   ! RB-1000SAD (Robobel Type):
   !pers tooldata tRB1000SAD_0   := [true,[[181.9,0,472.5],[0.866025,0,0.5,0]],[10,[31,0,260],[1,0,0,0],0,0,0]];
   !pers tooldata tRB1000SAD_100 := [true,[[268.5,0,522.5],[0.866025,0,0.5,0]],[10,[31,0,260],[1,0,0,0],0,0,0]];
   !pers tooldata tRB1000SAD_150 := [true,[[311.8,0,547.5],[0.866025,0,0.5,0]],[10,[31,0,260],[1,0,0,0],0,0,0]];
   !pers tooldata tRB1000SAD_200 := [true,[[355.1,0,572.5],[0.866025,0,0.5,0]],[10,[31,0,260],[1,0,0,0],0,0,0]];
   !pers tooldata tRB1000SAD_250 := [true,[[398.4,0,597.5],[0.866025,0,0.5,0]],[10,[31,0,260],[1,0,0,0],0,0,0]];
   !pers tooldata tRB1000SAD_300 := [true,[[441.7,0,622.5],[0.866025,0,0.5,0]],[10,[31,0,260],[1,0,0,0],0,0,0]];

   ! RB-1000SSD (Robobel Type):
   !PERS tooldata tRB1000SSD_0   := [true,[[181.9,0,472.5],[0.866025,0,0.5,0]],[10,[31,0,260],[1,0,0,0],0,0,0]];
   !PERS tooldata tRB1000SSD_100 := [true,[[268.5,0,522.5],[0.866025,0,0.5,0]],[10,[31,0,260],[1,0,0,0],0,0,0]];
   !PERS tooldata tRB1000SSD_150 := [true,[[311.8,0,547.5],[0.866025,0,0.5,0]],[10,[31,0,260],[1,0,0,0],0,0,0]];
   !PERS tooldata tRB1000SSD_200 := [true,[[355.1,0,572.5],[0.866025,0,0.5,0]],[10,[31,0,260],[1,0,0,0],0,0,0]];
   !PERS tooldata tRB1000SSD_250 := [true,[[398.4,0,597.5],[0.866025,0,0.5,0]],[10,[31,0,260],[1,0,0,0],0,0,0]];
   !PERS tooldata tRB1000SSD_300 := [true,[[441.7,0,622.5],[0.866025,0,0.5,0]],[10,[31,0,260],[1,0,0,0],0,0,0]];



   ! Speed data:
   const speeddata vPaint50   := [50,300,1000,50];
   const speeddata vPaint100  := [100,300,100,100];
   const speeddata vPaint150  := [150,300,150,150];
   const speeddata vPaint200  := [200,300,200,200];
   const speeddata vPaint250  := [250,300,250,250];
   const speeddata vPaint300  := [300,300,300,300];
   const speeddata vPaint350  := [350,300,350,350];
   const speeddata vPaint400  := [400,300,400,400];
   const speeddata vPaint450  := [450,300,450,450];
   const speeddata vPaint500  := [500,300,500,500];
   const speeddata vPaint550  := [550,300,1000,500];
   const speeddata vPaint600  := [600,300,1000,500];
   const speeddata vPaint650  := [650,300,1000,500];
   const speeddata vPaint700  := [700,300,1000,500];
   const speeddata vPaint750  := [750,300,1000,500];
   const speeddata vPaint800  := [800,300,1000,500];
   const speeddata vPaint850  := [850,300,1000,500];
   const speeddata vPaint900  := [900,300,1000,500];
   const speeddata vPaint950  := [950,300,1000,500];
   const speeddata vPaint1000 := [1000,300,1000,500];
   const speeddata vPaint1100 := [1100,300,1000,500];
   const speeddata vPaint1200 := [1200,300,1000,500];
   const speeddata vPaint1300 := [1300,300,1000,500];
   const speeddata vPaint1400 := [1400,300,1000,500];
   const speeddata vPaint1500 := [1500,300,1000,500];
   const speeddata vPaint1600 := [1600,300,1000,500];
   const speeddata vPaint1700 := [1700,300,1000,500];
   const speeddata vPaint1800 := [1800,300,1000,500];
   const speeddata vPaint1900 := [1900,300,1000,500];
   const speeddata vPaint2000 := [2000,300,1000,500];
   const speeddata vPaint2100 := [2100,300,1000,500];
   const speeddata vPaint2200 := [2200,300,1000,500];
   const speeddata vPaint2300 := [2300,300,1000,500];
   const speeddata vPaint2400 := [2400,300,1000,500];
   const speeddata vPaint2500 := [2500,300,1000,500];

   ! Speed data (High Flow Bell):
   const speeddata vHFB50   := [50,150,50,50];
   const speeddata vHFB100  := [100,150,100,100];
   const speeddata vHFB150  := [150,150,150,150];
   const speeddata vHFB200  := [200,150,200,200];
   const speeddata vHFB250  := [250,150,250,250];
   const speeddata vHFB300  := [300,150,300,300];
   const speeddata vHFB350  := [350,150,350,350];
   const speeddata vHFB400  := [400,150,400,400];
   const speeddata vHFB450  := [450,150,450,450];
   const speeddata vHFB500  := [500,150,500,500];
   const speeddata vHFB550  := [550,150,1000,500];
   const speeddata vHFB600  := [600,150,1000,500];
   const speeddata vHFB650  := [650,150,1000,500];
   const speeddata vHFB700  := [700,150,1000,500];
   const speeddata vHFB750  := [750,150,1000,500];
   const speeddata vHFB800  := [800,150,1000,500];
   const speeddata vHFB850  := [850,150,1000,500];
   const speeddata vHFB900  := [900,150,1000,500];
   const speeddata vHFB950  := [950,150,1000,500];
   const speeddata vHFB1000 := [1000,150,1000,500];
   const speeddata vHFB1100 := [1100,150,1000,500];
   const speeddata vHFB1200 := [1200,150,1000,500];
   const speeddata vHFB1300 := [1300,150,1000,500];
   const speeddata vHFB1400 := [1400,150,1000,500];
   const speeddata vHFB1500 := [1500,150,1000,500];
   const speeddata vHFB1600 := [1600,150,1000,500];
   const speeddata vHFB1700 := [1700,150,1000,500];
   const speeddata vHFB1800 := [1800,150,1000,500];
   const speeddata vHFB1900 := [1900,150,1000,500];
   const speeddata vHFB2000 := [2000,150,1000,500];
   const speeddata vHFB2100 := [2100,150,1000,500];
   const speeddata vHFB2200 := [2200,150,1000,500];
   const speeddata vHFB2300 := [2300,150,1000,500];
   const speeddata vHFB2400 := [2400,150,1000,500];
   const speeddata vHFB2500 := [2500,150,1000,500];



   ! Zone data:
   const zonedata zPaint1   := [false,1,1,1,0.15,1,0.15];
   const zonedata zPaint5   := [false,5,8,8,0.8,8,0.8];
   const zonedata zPaint10  := [false,10,15,15,1.5,15,1.5];
   const zonedata zPaint15  := [false,15,23,23,2.3,23,2.3];
   const zonedata zPaint20  := [false,20,30,30,3,30,3];
   const zonedata zPaint30  := [false,30,45,45,4.5,45,4.5];
   const zonedata zPaint40  := [false,40,60,60,6,60,6];
   const zonedata zPaint50  := [false,50,75,75,7.5,75,7.5];
   const zonedata zPaint60  := [false,60,90,90,9,90,9];
   const zonedata zPaint80  := [false,80,120,120,12,120,12];
   const zonedata zPaint100 := [false,100,150,150,15,150,15];
   const zonedata zPaint150 := [false,150,225,225,23,225,23];
   const zonedata zPaint200 := [false,200,300,300,30,300,30];
   const zonedata zPaint250 := [false,250,375,375,37.5,375,37.5];
   const zonedata zPaint300 := [false,300,450,450,45,450,45];



   proc ConfSettingsOff()
      ConfJ \Off;
      ConfL \Off;
   endproc



endmodule

--- Backups/Robo_open_v2/RAPID/TASK1/SYSMOD/sysdata.sys ---
module sysdata(sysmodule)

   ! Warning: Do not remove standard data from this module.

   pers robtarget pHomePos   := [[0,0,0],[9E+09,9E+09,9E+09,9E+09],[-1,-1,1,0],[9E+09,9E+09,9E+09,9E+09,9E+09,9E+09]];
   pers robtarget pMtrlChPos := [[0,0,0],[9E+09,9E+09,9E+09,9E+09],[-1,-1,1,0],[9E+09,9E+09,9E+09,9E+09,9E+09,9E+09]];
   pers robtarget pReadyPos  := [[0,0,0],[9E+09,9E+09,9E+09,9E+09],[-1,-1,1,0],[9E+09,9E+09,9E+09,9E+09,9E+09,9E+09]];
   pers robtarget pUserPos   := [[0,0,0],[9E+09,9E+09,9E+09,9E+09],[-1,-1,1,0],[9E+09,9E+09,9E+09,9E+09,9E+09,9E+09]];

   pers jointtarget jHomePos   := [[9E+09,9E+09,9E+09,9E+09,9E+09,9E+09],[9E+09,9E+09,9E+09,9E+09,9E+09,0]];
   pers jointtarget jMtrlChPos := [[9E+09,9E+09,9E+09,9E+09,9E+09,9E+09],[9E+09,9E+09,9E+09,9E+09,9E+09,0]];
   pers jointtarget jReadyPos  := [[9E+09,9E+09,9E+09,9E+09,9E+09,9E+09],[9E+09,9E+09,9E+09,9E+09,9E+09,0]];
   pers jointtarget jUserPos   := [[9E+09,9E+09,9E+09,9E+09,9E+09,9E+09],[9E+09,9E+09,9E+09,9E+09,9E+09,0]];

   pers tooldata tUserTool0 := [TRUE,[[0,0,0],[1,0,0,0]],[0.001,[0,0,0.001],[1,0,0,0],0,0,0]];

endmodule

--- Backups/Robo_open_v2/RAPID/TASK3/SYSMOD/custpnt.sys ---
module custpnt(sysmodule)



   proc InitCustPnt()
      !
      ! This will be executed during startup...
      !
      Subscribe TOGGLE_PATASK, "ToggleCustom";
   endproc



   proc ToggleCustom()
      !
      ! This will be executed on ProgramToggle or CommandToggle,
      ! depending on what IO interface is installed.
      !
      ! WARNING: Do not put time-consuming instructions here,
      ! since this is run in a trap, and will block the IO interface.
      !
   endproc



   proc Cmd1001(num nInparams{*}, string stInparams{*}, inout num nOutparams{*}, inout string stOutparams{*})
      !
      ! Insert RAPID code for command here...
      !
      nOutparams{1} := CMD_OK;
   error
      nOutparams{1} := CMD_FAILED;
      return;
   endproc



   proc Cmd1002(num nInparams{*}, string stInparams{*}, inout num nOutparams{*}, inout string stOutparams{*})
      !
      ! Insert RAPID code for command here...
      !
      nOutparams{1} := CMD_OK;
   error
      nOutparams{1} := CMD_FAILED;
      return;
   endproc



endmodule

--- Backups/Robo_open_v2/RAPID/TASK3/SYSMOD/qdata.sys ---
module qdata(sysmodule)



   pers num nJobQueueSize := 0; ! Actual number of entries/jobs.

   pers recJobInfo JobQueue{10} :=
      [[0,0,0,0,0,0,0,false],
       [0,0,0,0,0,0,0,false],
       [0,0,0,0,0,0,0,false],
       [0,0,0,0,0,0,0,false],
       [0,0,0,0,0,0,0,false],
       [0,0,0,0,0,0,0,false],
       [0,0,0,0,0,0,0,false],
       [0,0,0,0,0,0,0,false],
       [0,0,0,0,0,0,0,false],
       [0,0,0,0,0,0,0,false]];



endmodule

--- Backups/Robo_open_v2/HOME/programs/calpos.mod ---
module calpos

   ! SCOPE: Universal calibration/sync position program.

   proc mainCalPos()
      var jointtarget jLocalCalPos;

      ! Dummy instruction for SetPP.
      WaitTime 1;

      ! Set default values for all axis.
      jLocalCalPos := [[9E+09,9E+09,9E+09,9E+09,9E+09,9E+09],[9E+09,9E+09,9E+09,9E+09,9E+09,0]];

      jLocalCalPos.robax.rax_1 := nArmCalPos("rob1_1");
      jLocalCalPos.robax.rax_2 := nArmCalPos("rob1_2");
      jLocalCalPos.robax.rax_3 := nArmCalPos("rob1_3");
      jLocalCalPos.robax.rax_4 := nArmCalPos("rob1_4");
      jLocalCalPos.robax.rax_5 := nArmCalPos("rob1_5");
      jLocalCalPos.robax.rax_6 := nArmCalPos("rob1_6");

      if nRobSerialPart() = 5500 then
         ! IRB5500 has special values on axis 5 and 6, just set to 0 as stated in the manual.
         jLocalCalPos.robax.rax_5 := 0;
         jLocalCalPos.robax.rax_6 := 0;
      endif

      if stSingleJoint("AX7_1") <> "" then
         ! 7-axis robot.
         jLocalCalPos.extax.eax_a := nArmCalPos(stSingleJoint("AX7_1") \NoConversion);
      elseif nArmCalPos("obp_3") <> 9E+09 then
         ! 3-axis TurnTable.
         !IndReset OBP,2\RefNum:=0\Short;
         !IndReset OBP,3\RefNum:=0\Short;
         jLocalCalPos.extax.eax_a := nArmCalPos("obp_1");
         jLocalCalPos.extax.eax_b := nArmCalPos("obp_2");
         jLocalCalPos.extax.eax_c := nArmCalPos("obp_3");
      elseif nArmCalPos("obp_2") <> 9E+09 then
         ! 2-axis TurnTable.
         jLocalCalPos.extax.eax_a := nArmCalPos("obp_1");
         jLocalCalPos.extax.eax_b := nArmCalPos("obp_2");
      elseif nArmCalPos("obp_1") <> 9E+09 then
         ! 1-axis TurnTable.
         jLocalCalPos.extax.eax_a := nArmCalPos("obp_1");
      elseif nArmCalPos("track1") <> 9E+09 then
         ! IRB5350-02.
         jLocalCalPos.robax.rax_4 := 0;
         jLocalCalPos.robax.rax_5 := 0;
         jLocalCalPos.robax.rax_6 := 0;
         jLocalCalPos.extax.eax_a := nArmCalPos("track1" \NoConversion);
      else
         ! Attempt to get values for 8-axis robot.
         jLocalCalPos.extax.eax_a := nArmCalPos("rob1_7" \NoConversion);
         jLocalCalPos.extax.eax_b := nArmCalPos("rob1_8" \NoConversion);
      endif

      if stSingleJoint("H1AngleAxis") <> "" then
         ! Global CBS.
         jLocalCalPos.extax.eax_b := 0;
         jLocalCalPos.extax.eax_c := 0;
         jLocalCalPos.extax.eax_d := 0;
         jLocalCalPos.extax.eax_e := 0;
      endif

      MoveAbsJ jLocalCalPos,v100,fine,tool0;
      Stop;
   endproc

   local func num nArmCalPos(string stArm \switch NoConversion)
      var num nCalPos;
      ReadCfgData "/MOC/ARM/" + stArm, "cal_position", nCalPos;
      if Present(NoConversion) then
         return nCalPos;
      else
         return Round(nCalPos * (180 / 3.1415926) \Dec := 3);
      endif
   error
      if errno = ERR_CFG_NOTFND then
         SkipWarn;
         return 9E+09;
      endif
   endfunc

   local func string stSingleJoint(string stSingle)
      var string stJoint;
      ReadCfgData "/MOC/SINGLE/" + stSingle, "use_joint", stJoint;
      return stJoint;
   error
      if errno = ERR_CFG_NOTFND then
         SkipWarn;
         return "";
      endif
   endfunc

   local func num nRobSerialPart()
      var string stPart;
      var num nPart;
      ReadCfgData "/MOC/ROBOT_SERIAL_NUMBER/PID", "robot_serial_number_high_part", stPart;
      if StrToVal(StrPart(stPart, 1, StrFind(stPart, 1, "_") - 1), nPart) then
         return nPart;
      else
         return 9E+09;
      endif
   error
      SkipWarn;
      return 9E+09;
   endfunc

endmodule

--- Backups/Robo_open_v2/HOME/programs/m1.mod ---
MODULE M1

  PROC mainM1()
     WaitTime 10;
  ENDPROC
ENDMODULE

--- Backups/Robo_open_v2/HOME/programs/m10001.mod ---
module m10001

   ! SCOPE: Motion program for home position.

   proc mainm10001()
      if jHomePos.robax.rax_1 = 9E+09 then
         ErrWrite \W, "Home position not taught!", "";
      else
         MoveAbsJ jHomePos,v300,fine,tUserTool0;
      endif
   endproc

endmodule

--- Backups/Robo_open_v2/HOME/programs/m2.mod ---
MODULE M2

  PROC mainM2()
     WaitTime 10;
  ENDPROC
ENDMODULE

--- Backups/Robo_open_v2/HOME/programs/m3.mod ---
MODULE M3

  PROC mainM3()
     WaitTime 10;
  ENDPROC
ENDMODULE

--- Backups/Robot_ISEP_IRB140/SYSPAR/EIO.cfg ---
EIO:CFG_1.0:5:0::
#
EIO_BUS:

      -Name "Virtual1" -ConnectorID "SIM1"

      -Name "DeviceNet1" -BusType "DNET" -ConnectorID "PCI1"\
      -ConnectorLabel "First DeviceNet"
#
EIO_UNIT_TYPE:

      -Name "Virtual" -VendorName "ABB" -ProductName "Virtual unit"

      -Name "DN_GENERIC" -BusType "DNET" -DN_ExplicitMsgEnabled \
      -DN_C1OutputSize -1 -DN_C1InputSize -1

      -Name "d320" -BusType "DNET" -VendorName "ABB Robotics"\
      -ProductName "120 Vac Unit" -DN_VendorId 75 -DN_ProductCode 1\
      -DN_DeviceType 7 -DN_MajorRev 1 -DN_ExplicitMsgEnabled  -DN_C1Interval 50\
      -DN_C1OutputSize 2 -DN_C1InputSize 2

      -Name "d327A" -BusType "DNET" -VendorName "ABB Robotics"\
      -ProductName "Combi Unit" -DN_VendorId 75 -DN_ProductCode 2\
      -DN_DeviceType 100 -DN_MajorRev 5 -DN_ExplicitMsgEnabled  -DN_C1Type "COS"\
      -DN_C1OutputSize 6 -DN_C1InputSize 2

      -Name "d328A" -BusType "DNET" -VendorName "ABB Robotics"\
      -ProductName "24 VDC Unit" -DN_VendorId 75 -DN_ProductCode 3\
      -DN_DeviceType 7 -DN_ExplicitMsgEnabled  -DN_C1Type "COS"\
      -DN_C1OutputSize 2 -DN_C1InputSize 2

      -Name "d332A" -BusType "DNET" -VendorName "ABB Robotics"\
      -ProductName "Relay Unit" -DN_VendorId 75 -DN_ProductCode 5\
      -DN_DeviceType 7 -DN_MajorRev 2 -DN_ExplicitMsgEnabled  -DN_C1Type "COS"\
      -DN_C1OutputSize 2 -DN_C1InputSize 2

      -Name "d355A" -BusType "DNET" -VendorName "ABB Robotics"\
      -ProductName "Analog Unit" -DN_VendorId 75 -DN_ProductCode 10\
      -DN_DeviceType 100 -DN_MajorRev 1 -DN_ExplicitMsgEnabled \
      -DN_C1Interval 50 -DN_C1OutputSize 8 -DN_C1InputSize 8

      -Name "d651" -BusType "DNET" -VendorName "ABB Robotics"\
      -ProductName "Combi Unit" -DN_VendorId 75 -DN_ProductCode 25\
      -DN_DeviceType 100 -DN_ExplicitMsgEnabled  -DN_C1Type "COS"\
      -DN_C1OutputSize 5 -DN_C1InputSize 1

      -Name "d652" -BusType "DNET" -VendorName "ABB Robotics"\
      -ProductName "24 VDC Unit" -DN_VendorId 75 -DN_ProductCode 26\
      -DN_DeviceType 7 -DN_ExplicitMsgEnabled  -DN_C1Type "COS"\
      -DN_C1OutputSize 2 -DN_C1InputSize 2

      -Name "d653" -BusType "DNET" -VendorName "ABB Robotics"\
      -ProductName "Relay Unit" -DN_VendorId 75 -DN_ProductCode 27\
      -DN_DeviceType 7 -DN_ExplicitMsgEnabled  -DN_C1Type "COS"\
      -DN_C1OutputSize 1 -DN_C1InputSize 1

      -Name "DN_SLAVE" -BusType "DNET" -VendorName "ABB Robotics" -DN_VendorId 8\
      -DN_ProductCode 12 -DN_DeviceType 12 -DN_ExplicitMsgEnabled \
      -DN_C1Interval 50 -DN_C1OutputSize 8 -DN_C1InputSize 8

      -Name "DN_INTERNAL_SLAVE" -BusType "DNET" -VendorName "ABB Robotics"\
      -ProductName "Internal DeviceNet Slave" -InternalSlave  -DN_C1OutputSize 8\
      -DN_C1InputSize 8

      -Name "d350B" -BusType "DNET" -VendorName "ABB Robotics"\
      -ProductName "RIO Adapter" -DN_VendorId 75 -DN_ProductCode 6\
      -DN_DeviceType 7 -DN_MajorRev 2 -DN_ExplicitMsgEnabled  -DN_C1Type "COS"\
      -DN_C1OutputSize -1 -DN_C1InputSize -1

      -Name "DN_SLAVE_FA" -BusType "DNET" -VendorName "ABB Robotics"\
      -ProductName "DeviceNet Fieldbus Adapter Slave" -DN_VendorId 75\
      -DN_ProductCode 98 -DN_DeviceType 12 -DN_MajorRev 2 -DN_MinorRev 1\
      -DN_ExplicitMsgEnabled  -DN_C1Type "COS" -DN_C1OutputSize 8\
      -DN_C1InputSize 8

      -Name "d351A" -BusType "DNET" -VendorName "ABB Robotics"\
      -ProductName "IBS Adapter" -DN_VendorId 75 -DN_ProductCode 7\
      -DN_DeviceType 7 -DN_MajorRev 1 -DN_ExplicitMsgEnabled  -DN_C1Type "COS"\
      -DN_C1OutputSize -1 -DN_C1InputSize -1

      -Name "d352A" -BusType "DNET" -VendorName "ABB Robotics"\
      -ProductName "PBUS Adapter" -DN_VendorId 75 -DN_ProductCode 8\
      -DN_DeviceType 7 -DN_MajorRev 1 -DN_ExplicitMsgEnabled  -DN_C1Type "COS"\
      -DN_C1OutputSize -1 -DN_C1InputSize -1

      -Name "d352B" -BusType "DNET" -VendorName "ABB Robotics"\
      -ProductName "PBUS Adapter" -DN_VendorId 75 -DN_ProductCode 8\
      -DN_DeviceType 7 -DN_MajorRev 1 -DN_ExplicitMsgEnabled  -DN_C1Type "COS"\
      -DN_C1OutputSize -1 -DN_C1InputSize -1

      -Name "d378A" -BusType "DNET" -VendorName "ABB Robotics"\
      -ProductName "CCLink Adapter" -DN_VendorId 75 -DN_ProductCode 17\
      -DN_DeviceType 7 -DN_MajorRev 1 -DN_ExplicitMsgEnabled  -DN_C1Interval 50\
      -DN_C1OutputSize -1 -DN_C1InputSize -1
#
EIO_COMMAND_TYPE:

      -Name "LinkAddr" -UnitType "d350B" -DefValue "1" -OrderNr 1\
      -DN_Path "6,20 64 24 01 30 01,C6,1"

      -Name "DataRate" -UnitType "d350B" -DefValue "0" -OrderNr 2\
      -DN_Path "6,20 64 24 01 30 02,C6,1"

      -Name "StartQ" -UnitType "d350B" -DefValue "0" -OrderNr 3\
      -DN_Path "6,20 64 24 01 30 03,C6,1"

      -Name "RackSize" -UnitType "d350B" -DefValue "0" -OrderNr 4\
      -DN_Path "6,20 64 24 01 30 04,C6,1"

      -Name "LastRack" -UnitType "d350B" -DefValue "0" -OrderNr 5\
      -DN_Path "6,20 64 24 01 30 05,C1,1"

      -Name "D350Breset" -UnitType "d350B" -DefValue "0" -OrderNr 6\
      -DN_Path "4,20 01 24 01,C1,1" -DN_Service 5

      -Name "DataWidth" -UnitType "d351A" -DefValue "3" -OrderNr 1\
      -DN_Path "6,20 65 24 01 30 01,C6,1"

      -Name "D351Areset" -UnitType "d351A" -DefValue "0" -OrderNr 2\
      -DN_Path "4,20 01 24 01,C1,1" -DN_Service 5

      -Name "MasterInputSize" -UnitType "d352A" -DefValue "1" -OrderNr 1\
      -DN_Path "6,20 67 24 01 30 02,C6,1"

      -Name "MasterOutputSize" -UnitType "d352A" -DefValue "1" -OrderNr 2\
      -DN_Path "6,20 67 24 01 30 03,C6,1"

      -Name "StationAddress" -UnitType "d352A" -DefValue "126" -OrderNr 3\
      -DN_Path "6,20 67 24 01 30 04,C6,1"

      -Name "D352Areset" -UnitType "d352A" -DefValue "0" -OrderNr 4\
      -DN_Path "4,20 01 24 01,C1,1" -DN_Service 5

      -Name "MasterInputSize_B" -UnitType "d352B" -DefValue "1" -OrderNr 1\
      -DN_Path "6,20 67 24 01 30 02,C6,1"

      -Name "MasterOutputSize_B" -UnitType "d352B" -DefValue "1" -OrderNr 2\
      -DN_Path "6,20 67 24 01 30 03,C6,1"

      -Name "StationAddress_B" -UnitType "d352B" -DefValue "126" -OrderNr 3\
      -DN_Path "6,20 67 24 01 30 04,C6,1"

      -Name "D352Breset" -UnitType "d352B" -DefValue "0" -OrderNr 4\
      -DN_Path "4,20 01 24 01,C1,1" -DN_Service 5

      -Name "StationNo" -UnitType "d378A" -DefValue "1" -OrderNr 1\
      -DN_Path "6,20 68 24 01 30 01,C6,1"

      -Name "BaudRate" -UnitType "d378A" -DefValue "0" -OrderNr 2\
      -DN_Path "6,20 68 24 01 30 02,C6,1"

      -Name "OccStat" -UnitType "d378A" -DefValue "1" -OrderNr 3\
      -DN_Path "6,20 68 24 01 30 03,C6,1"

      -Name "BasicIO" -UnitType "d378A" -DefValue "0" -OrderNr 4\
      -DN_Path "6,20 68 24 01 30 04,C1,1"

      -Name "D378Areset" -UnitType "d378A" -DefValue "0" -OrderNr 5\
      -DN_Path "4,20 01 24 01,C1,1" -DN_Service 5
#
EIO_ACCESS:

      -Name "All" -Rapid  -LocalManual  -LocalAuto  -RemoteManual  -RemoteAuto

--- Backups/Robo_open_v2/SYSPAR/EIO.cfg ---
EIO:CFG_1.0:5:0::
#
EIO_BUS:

      -Name "Virtual1" -ConnectorID "SIM1"

      -Name "ICIBUS" -BusType "PIO" -ConnectorID "PIO2"\
      -ConnectorLabel "First ICI Bus"
#
EIO_UNIT_TYPE:

      -Name "Virtual" -VendorName "ABB" -ProductName "Virtual unit"

      -Name "ICI_TYPE" -BusType "PIO" -VendorName "ABB"\
      -ProductName "IPS (ICI) unit"
#
EIO_UNIT:

      -Name "PIB" -UnitType "ICI_TYPE" -Bus "ICIBUS"\
      -UnitLabel "Process Interface Board" -PIO_Address "192.168.126.200"

      -Name "PibSaf" -UnitType "ICI_TYPE" -Bus "ICIBUS" -UnitLabel "Safety Unit"\
      -PIO_Address "192.168.126.200"

      -Name "SysComm" -UnitType "Virtual" -Bus "Virtual1"

      -Name "CommandIO" -UnitType "Virtual" -Bus "Virtual1"

      -Name "DummyIO" -UnitType "Virtual" -Bus "Virtual1"
#
EIO_SIGNAL:

      -Name "sdoAutoOn" -SignalType "DO" -Unit "SysComm" -UnitMap "0"

      -Name "sdoCycleOn" -SignalType "DO" -Unit "SysComm" -UnitMap "1"

      -Name "sdoEmStop" -SignalType "DO" -Unit "SysComm" -UnitMap "2"

      -Name "sdoError" -SignalType "DO" -Unit "SysComm" -UnitMap "3"

      -Name "sdoMotOnState" -SignalType "DO" -Unit "SysComm" -UnitMap "4"

      -Name "sdoRunchOk" -SignalType "DO" -Unit "SysComm" -UnitMap "5"

      -Name "sdoMotorOn" -SignalType "DO" -Unit "SysComm" -UnitMap "6"

      -Name "sdoMotorOff" -SignalType "DO" -Unit "SysComm" -UnitMap "7"

      -Name "sdoStart" -SignalType "DO" -Unit "SysComm" -UnitMap "8"

      -Name "sdoStop" -SignalType "DO" -Unit "SysComm" -UnitMap "9"

      -Name "sdoResetError" -SignalType "DO" -Unit "SysComm" -UnitMap "10"

      -Name "sdoSysReset" -SignalType "DO" -Unit "SysComm" -UnitMap "11"

      -Name "sdoStartMain" -SignalType "DO" -Unit "SysComm" -UnitMap "12"

      -Name "sdoManRedSpeed" -SignalType "DO" -Unit "SysComm" -UnitMap "13"

      -Name "sdoManFullSpeed" -SignalType "DO" -Unit "SysComm" -UnitMap "14"

      -Name "sdoSwitchInAuto" -SignalType "DO" -Unit "SysComm" -UnitMap "15"

      -Name "doPntRapidError" -SignalType "DO" -Unit "SysComm" -UnitMap "20"

      -Name "doAutoMode" -SignalType "DO" -Unit "SysComm" -UnitMap "21"

      -Name "doInitialized" -SignalType "DO" -Unit "SysComm" -UnitMap "22"

      -Name "doInModule" -SignalType "DO" -Unit "SysComm" -UnitMap "23" -Store

      -Name "doJobInProgress" -SignalType "DO" -Unit "SysComm" -UnitMap "24"\
      -Store

      -Name "doQueueNotEmpty" -SignalType "DO" -Unit "SysComm" -UnitMap "25"

      -Name "doQueueFull" -SignalType "DO" -Unit "SysComm" -UnitMap "26"

      -Name "doQueueExpedited" -SignalType "DO" -Unit "SysComm" -UnitMap "27"

      -Name "doQueuePause" -SignalType "DO" -Unit "SysComm" -UnitMap "28"

      -Name "doSpyStart" -SignalType "DO" -Unit "SysComm" -UnitMap "29"\
      -Access "ALL"

      -Name "doSpyStop" -SignalType "DO" -Unit "SysComm" -UnitMap "30"\
      -Access "ALL"

      -Name "doMtrlSupOn" -SignalType "DO" -Unit "SysComm" -UnitMap "31"

      -Name "doHomePos" -SignalType "DO" -Unit "SysComm" -UnitMap "32"\
      -Access "INTERNAL"

      -Name "doMtrlChangePos" -SignalType "DO" -Unit "SysComm" -UnitMap "33"\
      -Access "INTERNAL"

      -Name "doReadyPos" -SignalType "DO" -Unit "SysComm" -UnitMap "34"\
      -Access "INTERNAL"

      -Name "doUserPos" -SignalType "DO" -Unit "SysComm" -UnitMap "35"\
      -Access "INTERNAL"

      -Name "doModeChangeAck" -SignalType "DO" -Unit "SysComm" -UnitMap "36"

      -Name "doExStart" -SignalType "DO" -Unit "SysComm" -UnitMap "37"

      -Name "doCmdReady" -SignalType "DO" -Unit "SysComm" -UnitMap "38"

      -Name "doCmdExecuting" -SignalType "DO" -Unit "SysComm" -UnitMap "39"

      -Name "doTPUCmdReady" -SignalType "DO" -Unit "SysComm" -UnitMap "40"

      -Name "doGUICmdReady" -SignalType "DO" -Unit "SysComm" -UnitMap "41"

      -Name "doIntCommand" -SignalType "DO" -Unit "SysComm" -UnitMap "42"

      -Name "doDirectModule" -SignalType "DO" -Unit "SysComm" -UnitMap "43"

      -Name "doMainInMC" -SignalType "DO" -Unit "SysComm" -UnitMap "44"

      -Name "doPLCCmdReady" -SignalType "DO" -Unit "SysComm" -UnitMap "45"

      -Name "doRapidError" -SignalType "DO" -Unit "SysComm" -UnitMap "46"

      -Name "doStartVClock" -SignalType "DO" -Unit "SysComm" -UnitMap "47"\
      -Access "ALL"

      -Name "doUpdateVClock" -SignalType "DO" -Unit "SysComm" -UnitMap "48"\
      -Access "ALL"

      -Name "doPaintBackup" -SignalType "DO" -Unit "SysComm" -UnitMap "49"\
      -Access "ALL"

      -Name "AutomaticMode" -SignalType "DO" -Unit "DummyIO" -UnitMap "0"\
      -Access "RAPIDONLY"

      -Name "MasterGranted" -SignalType "DO" -Unit "DummyIO" -UnitMap "1"\
      -Access "RAPIDONLY"

      -Name "RunChainClosed" -SignalType "DO" -Unit "DummyIO" -UnitMap "2"\
      -Access "RAPIDONLY"

      -Name "RobotError" -SignalType "DO" -Unit "DummyIO" -UnitMap "3"\
      -Access "RAPIDONLY"

      -Name "JobInProgress" -SignalType "DO" -Unit "DummyIO" -UnitMap "4"\
      -Access "RAPIDONLY"

      -Name "JobPending" -SignalType "DO" -Unit "DummyIO" -UnitMap "5"\
      -Access "RAPIDONLY"

      -Name "ReadyHighPri" -SignalType "DO" -Unit "DummyIO" -UnitMap "6"\
      -Access "RAPIDONLY"

      -Name "SystemRunning" -SignalType "DO" -Unit "DummyIO" -UnitMap "7"\
      -Access "RAPIDONLY"

      -Name "MtrlChRunning" -SignalType "DO" -Unit "DummyIO" -UnitMap "8"\
      -Access "RAPIDONLY"

      -Name "MtrlChangeOn" -SignalType "DO" -Unit "DummyIO" -UnitMap "9"\
      -Access "RAPIDONLY"

      -Name "MtrlSupplyEna" -SignalType "DO" -Unit "DummyIO" -UnitMap "10"\
      -Access "RAPIDONLY"

      -Name "MtrlSupplyError" -SignalType "DO" -Unit "DummyIO" -UnitMap "11"\
      -Access "RAPIDONLY"

      -Name "AppEnabled" -SignalType "DO" -Unit "DummyIO" -UnitMap "12"\
      -Access "RAPIDONLY"

      -Name "AppError" -SignalType "DO" -Unit "DummyIO" -UnitMap "13"\
      -Access "RAPIDONLY"

      -Name "HVEnabled" -SignalType "DO" -Unit "DummyIO" -UnitMap "14"\
      -Access "RAPIDONLY"

      -Name "HVError" -SignalType "DO" -Unit "DummyIO" -UnitMap "15"\
      -Access "RAPIDONLY"

      -Name "HeartBeat" -SignalType "DO" -Unit "DummyIO" -UnitMap "16"\
      -Access "RAPIDONLY"

      -Name "ConveyorHoldReq" -SignalType "DO" -Unit "DummyIO" -UnitMap "17"\
      -Access "RAPIDONLY"

      -Name "PotLifeTimeOut" -SignalType "DO" -Unit "DummyIO" -UnitMap "18"\
      -Access "RAPIDONLY"

      -Name "HomePos" -SignalType "DO" -Unit "DummyIO" -UnitMap "19"\
      -Access "RAPIDONLY"

      -Name "MtrlChangePos" -SignalType "DO" -Unit "DummyIO" -UnitMap "20"\
      -Access "RAPIDONLY"

      -Name "ReadyPos" -SignalType "DO" -Unit "DummyIO" -UnitMap "21"\
      -Access "RAPIDONLY"

      -Name "UserPos" -SignalType "DO" -Unit "DummyIO" -UnitMap "22"\
      -Access "RAPIDONLY"

      -Name "ReposFinished" -SignalType "DO" -Unit "DummyIO" -UnitMap "23"\
      -Access "RAPIDONLY"

      -Name "EmergencyStop" -SignalType "DO" -Unit "DummyIO" -UnitMap "24"\
      -Access "RAPIDONLY"

      -Name "JobComplete" -SignalType "DO" -Unit "DummyIO" -UnitMap "25"\
      -Access "RAPIDONLY"

      -Name "ManualMode" -SignalType "DO" -Unit "DummyIO" -UnitMap "26"\
      -Access "RAPIDONLY"

      -Name "ReadyToReceive" -SignalType "DO" -Unit "DummyIO" -UnitMap "27"\
      -Access "RAPIDONLY"

      -Name "MotorOn" -SignalType "DO" -Unit "DummyIO" -UnitMap "28"\
      -Access "RAPIDONLY"

      -Name "ProgramAck" -SignalType "DO" -Unit "DummyIO" -UnitMap "30"\
      -Access "RAPIDONLY"

      -Name "ProgramLoaded" -SignalType "DO" -Unit "DummyIO" -UnitMap "31"\
      -Access "RAPIDONLY"

      -Name "InModule" -SignalType "DO" -Unit "DummyIO" -UnitMap "69"\
      -Access "RAPIDONLY"

      -Name "ObjConnected" -SignalType "DO" -Unit "DummyIO" -UnitMap "70"\
      -Access "RAPIDONLY"

      -Name "ConveyorRunning" -SignalType "DO" -Unit "DummyIO" -UnitMap "71"\
      -Access "RAPIDONLY"

      -Name "CBSMotorOn" -SignalType "DO" -Unit "DummyIO" -UnitMap "72"\
      -Access "RAPIDONLY"

      -Name "PotLifeWarning" -SignalType "DO" -Unit "DummyIO" -UnitMap "73"\
      -Access "RAPIDONLY"

      -Name "GoingToAuto" -SignalType "DO" -Unit "DummyIO" -UnitMap "74"\
      -Access "RAPIDONLY"

      -Name "diModeChangeAck" -SignalType "DI" -Unit "SysComm" -UnitMap "1"

      -Name "A1Enable" -SignalType "DO" -Unit "SysComm" -UnitMap "100"\
      -Access "ALL"

      -Name "A1Error" -SignalType "DO" -Unit "SysComm" -UnitMap "101"\
      -Access "ALL"

      -Name "A1Material" -SignalType "GO" -Unit "SysComm" -UnitMap "110-119"\
      -Access "ALL"

      -Name "A1Brush" -SignalType "GO" -Unit "SysComm" -UnitMap "120-129"\
      -Access "ALL"

      -Name "A1BrushTabNdx" -SignalType "GO" -Unit "SysComm" -UnitMap "130-139"\
      -Access "ALL"

      -Name "A1Fluid" -SignalType "AO" -Unit "SysComm" -UnitMap "140-149"\
      -Access "ALL"

      -Name "A1HVErrNo" -SignalType "GO" -Unit "SysComm" -UnitMap "150-151"\
      -Access "ALL"

      -Name "A1HVEn" -SignalType "DO" -Unit "SysComm" -UnitMap "155"\
      -Access "ALL"

      -Name "SW_MOTOR_ON" -SignalType "DO" -Unit "PibSaf"\
      -UnitMap "Safety/OutPort1:SW_MOTOR_ON" -Access "INTERNAL"

      -Name "ReadyForMotorOn" -SignalType "DI" -Unit "PibSaf"\
      -UnitMap "Safety/InPort8:ReadyForMotorOn"

      -Name "MotorIsOn" -SignalType "DI" -Unit "PibSaf"\
      -UnitMap "Safety/InPort8:MotorIsOn"
#
EIO_CROSS:

      -Res "diModeChangeAck" -Act1 "doModeChangeAck"

      -Res "sdoManRedSpeed" -Act1 "MAN1" -Oper1 "AND" -Act2 "MAN2"

      -Res "sdoManFullSpeed" -Act1 "MANFS1" -Oper1 "AND" -Act2 "MANFS2"

      -Res "sdoSwitchInAuto" -Act1 "AUTO1" -Oper1 "AND" -Act2 "AUTO2"

      -Res "doAutoMode" -Act1 "sdoAutoOn" -Oper1 "AND" -Act2 "doInitialized"

      -Res "RobotError" -Act1 "sdoError" -Oper1 "OR" -Act2 "doPntRapidError"

      -Res "ReadyHighPri" -Act1 "sdoCycleOn" -Oper1 "AND"\
      -Act2 "doJobInProgress" -Act2_invert

      -Res "SystemRunning" -Act1 "sdoCycleOn" -Oper1 "AND" -Act2 "doQueuePause"\
      -Act2_invert

      -Res "doCmdReady" -Act1 "doPLCCmdReady" -Oper1 "OR" -Act2 "doTPUCmdReady"\
      -Oper2 "OR" -Act3 "doGUICmdReady" -Oper3 "OR" -Act4 "doIntCommand"

      -Res "AutomaticMode" -Act1 "doAutoMode"

      -Res "JobInProgress" -Act1 "doJobInProgress"

      -Res "JobPending" -Act1 "doQueueNotEmpty"

      -Res "EmergencyStop" -Act1 "sdoEmStop"

      -Res "MtrlSupplyEna" -Act1 "doMtrlSupOn"

      -Res "HomePos" -Act1 "doHomePos"

      -Res "MtrlChangePos" -Act1 "doMtrlChangePos"

      -Res "ReadyPos" -Act1 "doReadyPos"

      -Res "UserPos" -Act1 "doUserPos"

      -Res "AppEnabled" -Act1 "A1Enable"

      -Res "AppError" -Act1 "A1Error"

      -Res "A1HVEn" -Act1 "HVEnabled"

      -Res "InModule" -Act1 "doInModule"

      -Res "ManualMode" -Act1 "sdoManRedSpeed" -Oper1 "OR"\
      -Act2 "sdoManFullSpeed"

      -Res "ReadyToReceive" -Act1 "doInitialized" -Oper1 "AND"\
      -Act2 "doQueueFull" -Act2_invert

      -Res "GoingToAuto" -Act1 "sdoSwitchInAuto" -Oper1 "AND" -Act2 "sdoAutoOn"\
      -Act2_invert

      -Res "SW_MOTOR_ON" -Act1 "sdoMotorOn"

      -Res "RunChainClosed" -Act1 "ReadyForMotorOn"

      -Res "MotorOn" -Act1 "MotorIsOn"
#
EIO_ACCESS:

      -Name "All" -Rapid  -LocalManual  -LocalAuto  -RemoteManual  -RemoteAuto

      -Name "RAPIDONLY" -Rapid
#
SYSSIG_OUT:

      -Status "AutoOn" -Signal "sdoAutoOn"

      -Status "CycleOn" -Signal "sdoCycleOn"

      -Status "EmStop" -Signal "sdoEmStop"

      -Status "Error" -Signal "sdoError"

      -Status "MotOnState" -Signal "sdoMotOnState"

      -Status "RunchOk" -Signal "sdoRunchOk"
#
SYSSIG_IN:

      -Signal "sdoMotorOn" -Action "MotorOn"

      -Signal "sdoMotorOff" -Action "MotorOff"

      -Signal "sdoStart" -Action "Start"

      -Signal "sdoStop" -Action "Stop"

      -Signal "sdoResetError" -Action "ResetError"

      -Signal "sdoSysReset" -Action "SysReset"

      -Signal "sdoStartMain" -Action "StartMain"

      -Signal "doModeChangeAck" -Action "AckAutoMode"

--- Backups/Robo_open_v2/SYSPAR/PROC.cfg ---
PROC:CFG_1.0:5:0::
#
PW_SYSTEM:

      -name "PW_SYS" -pw_function "PW_FUNC"
#
PW_FUNCTION:

      -name "PW_FUNC" -do_repos_finished "ReposFinished"
